(* Logix 5000 project; controller MyFirstProject vendor 1 type 14 code 164 rev 33.11; software revision 33.01 *)

TASK MainTask (periodic, rate 250 ms, priority 10, watchdog 1000 ms) : MainProgram

MODULES
   Local : vendor 1 type 14 code 164 (ICP 0, rev 33.11)
END_MODULES

TYPE Motor :
STRUCT
   Power : REAL;
   Speed : INT;
   CmdOffOn : BOOL;
   SetSpeed : INT;
   Status : BOOL;
END_STRUCT
END_TYPE

TYPE MyDataType :
STRUCT
   PropertyTag1 : DINT;
   PropertyTag2 : DINT;
   Tag3 : DINT;
END_STRUCT
END_TYPE

TYPE Spindle :
STRUCT
   current : INT;
   speed : INT;
   status : BOOL;
END_STRUCT
END_TYPE

TYPE TankUDT :
STRUCT
   ValveInStatus : BOOL;
   ValveInCmd : BOOL;
   ValveOutStatus : BOOL;
   ValveOutCmd : BOOL;
   Level : REAL;
   SetPoint : REAL;
END_STRUCT
END_TYPE

VAR_GLOBAL   (* controller tags *)
   Motors : Motor[5] := ([0].Power := -0.2, [0].Speed := -1, [0].SetSpeed := 100, [1].Power := -0.2, [1].Speed := -1, [1].SetSpeed := 120, [2].Power := -0.2, [2].Speed := -1, [2].SetSpeed := 140, [3].Power := -0.2, [3].Speed := -1, [3].SetSpeed := 160, [4].Power := -0.2, [4].Speed := -1, [4].SetSpeed := 180);
   MyTag1 : MyDataType;
   SpindleArray : Spindle[10];
   Tank1 : TankUDT := (ValveInCmd := 1, Level := 49.0, SetPoint := 50.0);
   Tank2 : TankUDT := (ValveInCmd := 1, Level := 49.0, SetPoint := 50.0);
   TestBoolTag : BOOL := 1;
   TestIncrementTag : DINT := 58;
END_VAR

PROGRAM MainProgram   (* main routine Test *)
VAR
   Count : INT := 5;
   Direction : BOOL := 1;
   Init : BOOL := 1;
END_VAR

ROUTINE MainRoutine   (* ladder *)
END_ROUTINE

ROUTINE Test   (* structured text *)
   //Init Motors and WaterTank
   if (not Init) then
   	Init := 1;
   	Motors[0].SetSpeed := 100;
   	Motors[1].SetSpeed := 120;
   	Motors[2].SetSpeed := 140;
   	Motors[3].SetSpeed := 160;
   	Motors[4].SetSpeed := 180;
   	Tank2.SetPoint := 50.0;
   	Tank1.SetPoint := 50.0;
   	Tank2.Level := 1;
   	Tank1.Level := 1;
   end_if;
   
   if (TestIncrementTag = 0) then
   	Direction := 1;
   end_if;
   if (TestIncrementTag = 100) then
   	Direction := 0;
   end_if;
   if (TestBoolTag) then
   	if (Direction) then
   		TestIncrementTag := TestIncrementTag + 1;
   	else
   		TestIncrementTag := TestIncrementTag - 1;
   	end_if;
   end_if;
   
   //Tank 2 Logic
   if (Tank2.ValveInCmd) then
   	if (Tank2.Level < (Tank2.SetPoint -2)) then
   		Tank2.ValveInStatus := 1;
   		Tank2.Level := Tank2.Level + 3;
   	else
   		Tank2.ValveInStatus := 0;
   	end_if;
   else
   	Tank2.ValveInStatus := 0;
   end_if;
   
   if (Tank2.ValveOutCmd) then
   	if (Tank2.Level >= 3)  then
   		Tank2.ValveOutStatus := 1;
   		Tank2.Level := Tank2.Level - 3;
   	else
   		Tank2.ValveOutStatus := 0;
   	end_if;
   else
   	Tank2.ValveOutStatus := 0;
   end_if;
   
   //Tank 1 Logic
   if (Tank1.ValveInCmd) then
   	if (Tank1.Level < (Tank1.SetPoint -2)) then
   		Tank1.ValveInStatus := 1;
   		Tank1.Level := Tank1.Level + 3;
   	else
   		Tank1.ValveInStatus := 0;
   	end_if;
   else
   	Tank1.ValveInStatus := 0;
   end_if;
   
   if (Tank1.ValveOutCmd) then
   	if (Tank1.Level >= 3) then
   		Tank1.ValveOutStatus := 1;
   		Tank1.Level := Tank1.Level - 3;
   	else
   		Tank1.ValveOutStatus := 0;
   	end_if;
   else
   	Tank1.ValveOutStatus := 0;
   end_if;
   
   //Motor Logic
   for Count := 0 to 4 do
   	if (Motors[Count].CmdOffOn) then
   		Motors[Count].Status := 1;
   		if (Motors[Count].Speed <= Motors[Count].SetSpeed) then
   			Motors[Count].Speed := Motors[Count].Speed + 1;
   			Motors[Count].Power := Motors[Count].Power + 0.2;
   		end_if;
   	else
   		Motors[Count].Status := 0;
   		if (Motors[Count].Speed >= 0) then
   			Motors[Count].Speed := Motors[Count].Speed - 1;
   			Motors[Count].Power := Motors[Count].Power - 0.2;
   		end_if;
   	end_if;
   end_for;
   
END_ROUTINE
END_PROGRAM
